  PROC DrawPart23()
    MoveL Offs(pOrigin,149.54,33.47,0.00),v40,z0,tPen\WObj:=wPaper;
    MoveL Offs(pOrigin,149.54,33.47,0.00),v40,z0,tPen\WObj:=wPaper;
    MoveL Offs(pOrigin,150.93,34.68,0.00),v40,z0,tPen\WObj:=wPaper;
    MoveL Offs(pOrigin,156.56,36.34,0.00),v40,fine,tPen\WObj:=wPaper;
    MoveL Offs(pOrigin,156.56,36.34,6.00),v60,z5,tPen\WObj:=wPaper;
    MoveL Offs(pOrigin,156.88,32.94,6.00),vTravel,z5,tPen\WObj:=wPaper;
    MoveL Offs(pOrigin,156.88,32.94,0.00),v60,z0,tPen\WObj:=wPaper;
    MoveL Offs(pOrigin,160.17,29.65,0.00),v40,z0,tPen\WObj:=wPaper;
    MoveL Offs(pOrigin,160.49,29.76,0.00),v40,z0,tPen\WObj:=wPaper;
    MoveL Offs(pOrigin,161.44,27.63,0.00),v40,z0,tPen\WObj:=wPaper;
    MoveL Offs(pOrigin,162.08,23.81,0.00),v40,z0,tPen\WObj:=wPaper;
    MoveL Offs(pOrigin,161.76,20.62,0.00),v40,z0,tPen\WObj:=wPaper;
    MoveL Offs(pOrigin,160.98,18.60,0.00),v40,z0,tPen\WObj:=wPaper;
    MoveL Offs(pOrigin,157.73,17.25,0.00),v40,z0,tPen\WObj:=wPaper;
    MoveL Offs(pOrigin,156.98,16.40,0.00),v40,z0,tPen\WObj:=wPaper;
    MoveL Offs(pOrigin,153.37,15.41,0.00),v40,z0,tPen\WObj:=wPaper;
    MoveL Offs(pOrigin,148.59,15.09,0.00),v40,z0,tPen\WObj:=wPaper;
    MoveL Offs(pOrigin,147.21,15.41,0.00),v40,fine,tPen\WObj:=wPaper;
    MoveL Offs(pOrigin,147.21,15.41,6.00),v60,z5,tPen\WObj:=wPaper;
    MoveL Offs(pOrigin,149.01,16.79,6.00),vTravel,z5,tPen\WObj:=wPaper;
    MoveL Offs(pOrigin,149.01,16.79,0.00),v60,z0,tPen\WObj:=wPaper;
    MoveL Offs(pOrigin,146.99,15.41,0.00),v40,z0,tPen\WObj:=wPaper;
    MoveL Offs(pOrigin,142.43,14.35,0.00),v40,z0,tPen\WObj:=wPaper;
    MoveL Offs(pOrigin,138.39,14.39,0.00),v40,z0,tPen\WObj:=wPaper;
    MoveL Offs(pOrigin,137.43,15.52,0.00),v40,z0,tPen\WObj:=wPaper;
    MoveL Offs(pOrigin,136.79,17.54,0.00),v40,z0,tPen\WObj:=wPaper;
    MoveL Offs(pOrigin,136.79,17.54,0.00),v40,z0,tPen\WObj:=wPaper;
    MoveL Offs(pOrigin,141.47,19.31,0.00),v40,z0,tPen\WObj:=wPaper;
    MoveL Offs(pOrigin,142.96,20.19,0.00),v40,z0,tPen\WObj:=wPaper;
    MoveL Offs(pOrigin,142.96,20.19,0.00),v40,z0,tPen\WObj:=wPaper;
    MoveL Offs(pOrigin,143.91,20.37,0.00),v40,z0,tPen\WObj:=wPaper;
    MoveL Offs(pOrigin,144.12,20.73,0.00),v40,z0,tPen\WObj:=wPaper;
    MoveL Offs(pOrigin,144.23,20.73,0.00),v40,z0,tPen\WObj:=wPaper;
    MoveL Offs(pOrigin,145.40,21.19,0.00),v40,z0,tPen\WObj:=wPaper;
    MoveL Offs(pOrigin,145.82,22.21,0.00),v40,z0,tPen\WObj:=wPaper;
    MoveL Offs(pOrigin,144.80,25.29,0.00),v40,z0,tPen\WObj:=wPaper;
    MoveL Offs(pOrigin,143.81,25.61,0.00),v40,z0,tPen\WObj:=wPaper;
    MoveL Offs(pOrigin,142.21,25.01,0.00),v40,z0,tPen\WObj:=wPaper;
    MoveL Offs(pOrigin,141.89,24.55,0.00),v40,z0,tPen\WObj:=wPaper;
    MoveL Offs(pOrigin,142.99,20.94,0.00),v40,z0,tPen\WObj:=wPaper;
    MoveL Offs(pOrigin,144.23,20.73,0.00),v40,z0,tPen\WObj:=wPaper;
    MoveL Offs(pOrigin,143.70,21.79,0.00),v40,z0,tPen\WObj:=wPaper;
    MoveL Offs(pOrigin,142.74,24.12,0.00),v40,z0,tPen\WObj:=wPaper;
    MoveL Offs(pOrigin,144.23,24.87,0.00),v40,fine,tPen\WObj:=wPaper;
    MoveL Offs(pOrigin,144.23,24.87,6.00),v60,z5,tPen\WObj:=wPaper;
    MoveL Offs(pOrigin,144.98,23.38,6.00),vTravel,z5,tPen\WObj:=wPaper;
    MoveL Offs(pOrigin,144.98,23.38,0.00),v60,z0,tPen\WObj:=wPaper;
    MoveL Offs(pOrigin,145.05,22.21,0.00),v40,z0,tPen\WObj:=wPaper;
    MoveL Offs(pOrigin,144.23,22.00,0.00),v40,fine,tPen\WObj:=wPaper;
    MoveL Offs(pOrigin,144.23,22.00,6.00),v60,z5,tPen\WObj:=wPaper;
    MoveL Offs(pOrigin,145.51,21.15,6.00),vTravel,z5,tPen\WObj:=wPaper;
    MoveL Offs(pOrigin,145.51,21.15,0.00),v60,z0,tPen\WObj:=wPaper;
    MoveL Offs(pOrigin,147.21,21.68,0.00),v40,fine,tPen\WObj:=wPaper;
    MoveL Offs(pOrigin,147.21,21.68,6.00),v60,z5,tPen\WObj:=wPaper;
    MoveL Offs(pOrigin,144.34,26.78,6.00),vTravel,z5,tPen\WObj:=wPaper;
    MoveL Offs(pOrigin,144.34,26.78,0.00),v60,z0,tPen\WObj:=wPaper;
    MoveL Offs(pOrigin,141.68,25.90,0.00),v40,z0,tPen\WObj:=wPaper;
    MoveL Offs(pOrigin,141.04,25.40,0.00),v40,z0,tPen\WObj:=wPaper;
    MoveL Offs(pOrigin,141.04,25.40,0.00),v40,z0,tPen\WObj:=wPaper;
    MoveL Offs(pOrigin,141.89,24.87,0.00),v40,z0,tPen\WObj:=wPaper;
    MoveL Offs(pOrigin,141.04,25.40,0.00),v40,z0,tPen\WObj:=wPaper;
    MoveL Offs(pOrigin,138.39,24.69,0.00),v40,z0,tPen\WObj:=wPaper;
    MoveL Offs(pOrigin,130.31,20.76,0.00),v40,z0,tPen\WObj:=wPaper;
    MoveL Offs(pOrigin,127.55,18.92,0.00),v40,z0,tPen\WObj:=wPaper;
    MoveL Offs(pOrigin,127.34,18.39,0.00),v40,z0,tPen\WObj:=wPaper;
    MoveL Offs(pOrigin,127.34,18.39,0.00),v40,z0,tPen\WObj:=wPaper;
    MoveL Offs(pOrigin,127.44,17.64,0.00),v40,z0,tPen\WObj:=wPaper;
    MoveL Offs(pOrigin,128.72,16.79,0.00),v40,z0,tPen\WObj:=wPaper;
    MoveL Offs(pOrigin,132.12,16.69,0.00),v40,z0,tPen\WObj:=wPaper;
    MoveL Offs(pOrigin,135.94,17.22,0.00),v40,z0,tPen\WObj:=wPaper;
    MoveL Offs(pOrigin,135.94,17.22,0.00),v40,z0,tPen\WObj:=wPaper;
    MoveL Offs(pOrigin,136.16,17.54,0.00),v40,z0,tPen\WObj:=wPaper;
    MoveL Offs(pOrigin,136.79,17.54,0.00),v40,z0,tPen\WObj:=wPaper;
    MoveL Offs(pOrigin,136.90,16.37,0.00),v40,z0,tPen\WObj:=wPaper;
    MoveL Offs(pOrigin,117.14,11.48,0.00),v40,z0,tPen\WObj:=wPaper;
    MoveL Offs(pOrigin,106.30,12.44,0.00),v40,z0,tPen\WObj:=wPaper;
    MoveL Offs(pOrigin,105.98,12.76,0.00),v40,z0,tPen\WObj:=wPaper;
    MoveL Offs(pOrigin,105.03,12.86,0.00),v40,z0,tPen\WObj:=wPaper;
    MoveL Offs(pOrigin,104.71,13.18,0.00),v40,z0,tPen\WObj:=wPaper;
    MoveL Offs(pOrigin,104.28,12.97,0.00),v40,z0,tPen\WObj:=wPaper;
    MoveL Offs(pOrigin,105.03,12.86,0.00),v40,z0,tPen\WObj:=wPaper;
    MoveL Offs(pOrigin,105.77,12.76,0.00),v40,z0,tPen\WObj:=wPaper;
    MoveL Offs(pOrigin,107.57,13.39,0.00),v40,z0,tPen\WObj:=wPaper;
    MoveL Offs(pOrigin,124.15,16.90,0.00),v40,z0,tPen\WObj:=wPaper;
    MoveL Offs(pOrigin,125.21,17.54,0.00),v40,z0,tPen\WObj:=wPaper;
    MoveL Offs(pOrigin,125.21,17.54,0.00),v40,z0,tPen\WObj:=wPaper;
    MoveL Offs(pOrigin,122.88,18.21,0.00),v40,z0,tPen\WObj:=wPaper;
    MoveL Offs(pOrigin,122.34,19.88,0.00),v40,fine,tPen\WObj:=wPaper;
    MoveL Offs(pOrigin,122.34,19.88,6.00),v60,z5,tPen\WObj:=wPaper;
    MoveL Offs(pOrigin,123.09,21.15,6.00),vTravel,z5,tPen\WObj:=wPaper;
    MoveL Offs(pOrigin,123.09,21.15,0.00),v60,z0,tPen\WObj:=wPaper;
    MoveL Offs(pOrigin,123.51,21.58,0.00),v40,z0,tPen\WObj:=wPaper;
    MoveL Offs(pOrigin,123.09,21.15,0.00),v40,fine,tPen\WObj:=wPaper;
    MoveL Offs(pOrigin,123.09,21.15,6.00),v60,z5,tPen\WObj:=wPaper;
    MoveL Offs(pOrigin,124.57,22.42,6.00),vTravel,z5,tPen\WObj:=wPaper;
    MoveL Offs(pOrigin,124.57,22.42,0.00),v60,z0,tPen\WObj:=wPaper;
    MoveL Offs(pOrigin,125.00,22.85,0.00),v40,z0,tPen\WObj:=wPaper;
    MoveL Offs(pOrigin,124.57,22.42,0.00),v40,fine,tPen\WObj:=wPaper;
    MoveL Offs(pOrigin,124.57,22.42,6.00),v60,z5,tPen\WObj:=wPaper;
    MoveL Offs(pOrigin,121.07,22.32,6.00),vTravel,z5,tPen\WObj:=wPaper;
    MoveL Offs(pOrigin,121.07,22.32,0.00),v60,z0,tPen\WObj:=wPaper;
    MoveL Offs(pOrigin,119.37,22.42,0.00),v40,fine,tPen\WObj:=wPaper;
    MoveL Offs(pOrigin,119.37,22.42,6.00),v60,z5,tPen\WObj:=wPaper;
    MoveL Offs(pOrigin,112.99,23.70,6.00),vTravel,z5,tPen\WObj:=wPaper;
    MoveL Offs(pOrigin,112.99,23.70,0.00),v60,z0,tPen\WObj:=wPaper;
    MoveL Offs(pOrigin,111.82,24.23,0.00),v40,z0,tPen\WObj:=wPaper;
    MoveL Offs(pOrigin,112.36,24.76,0.00),v40,z0,tPen\WObj:=wPaper;
    MoveL Offs(pOrigin,111.61,24.27,0.00),v40,z0,tPen\WObj:=wPaper;
    MoveL Offs(pOrigin,109.70,25.01,0.00),v40,z0,tPen\WObj:=wPaper;
    MoveL Offs(pOrigin,107.93,26.36,0.00),v40,z0,tPen\WObj:=wPaper;
    MoveL Offs(pOrigin,106.72,28.48,0.00),v40,z0,tPen\WObj:=wPaper;
    MoveL Offs(pOrigin,106.72,28.48,0.00),v40,z0,tPen\WObj:=wPaper;
    MoveL Offs(pOrigin,100.88,31.49,0.00),v40,z0,tPen\WObj:=wPaper;
    MoveL Offs(pOrigin,93.44,33.86,0.00),v40,z0,tPen\WObj:=wPaper;
    MoveL Offs(pOrigin,91.85,34.75,0.00),v40,fine,tPen\WObj:=wPaper;
    MoveL Offs(pOrigin,91.85,34.75,6.00),v60,z5,tPen\WObj:=wPaper;
    MoveL Offs(pOrigin,90.79,28.59,6.00),vTravel,z5,tPen\WObj:=wPaper;
    MoveL Offs(pOrigin,90.79,28.59,0.00),v60,z0,tPen\WObj:=wPaper;
    MoveL Offs(pOrigin,94.61,26.67,0.00),v40,z0,tPen\WObj:=wPaper;
    MoveL Offs(pOrigin,94.61,26.67,0.00),v40,z0,tPen\WObj:=wPaper;
  ENDPROC

  PROC DrawPart24()
    MoveL Offs(pOrigin,94.08,25.19,0.00),v40,z0,tPen\WObj:=wPaper;
    MoveL Offs(pOrigin,94.08,25.19,0.00),v40,z0,tPen\WObj:=wPaper;
    MoveL Offs(pOrigin,95.04,24.87,0.00),v40,z0,tPen\WObj:=wPaper;
    MoveL Offs(pOrigin,95.04,24.87,0.00),v40,z0,tPen\WObj:=wPaper;
    MoveL Offs(pOrigin,95.57,26.36,0.00),v40,z0,tPen\WObj:=wPaper;
    MoveL Offs(pOrigin,95.57,26.36,0.00),v40,z0,tPen\WObj:=wPaper;
    MoveL Offs(pOrigin,104.49,23.91,0.00),v40,z0,tPen\WObj:=wPaper;
    MoveL Offs(pOrigin,104.81,23.59,0.00),v40,fine,tPen\WObj:=wPaper;
    MoveL Offs(pOrigin,104.81,23.59,6.00),v60,z5,tPen\WObj:=wPaper;
    MoveL Offs(pOrigin,109.06,23.27,6.00),vTravel,z5,tPen\WObj:=wPaper;
    MoveL Offs(pOrigin,109.06,23.27,0.00),v60,z0,tPen\WObj:=wPaper;
    MoveL Offs(pOrigin,109.59,24.98,0.00),v40,fine,tPen\WObj:=wPaper;
    MoveL Offs(pOrigin,109.59,24.98,6.00),v60,z5,tPen\WObj:=wPaper;
    MoveL Offs(pOrigin,117.56,29.54,6.00),vTravel,z5,tPen\WObj:=wPaper;
    MoveL Offs(pOrigin,117.56,29.54,0.00),v60,z0,tPen\WObj:=wPaper;
    MoveL Offs(pOrigin,113.31,35.49,0.00),v40,z0,tPen\WObj:=wPaper;
    MoveL Offs(pOrigin,113.42,36.13,0.00),v40,z0,tPen\WObj:=wPaper;
    MoveL Offs(pOrigin,115.44,35.53,0.00),v40,z0,tPen\WObj:=wPaper;
    MoveL Offs(pOrigin,117.67,34.11,0.00),v40,fine,tPen\WObj:=wPaper;
    MoveL Offs(pOrigin,117.67,34.11,6.00),v60,z5,tPen\WObj:=wPaper;
    MoveL Offs(pOrigin,118.41,39.00,6.00),vTravel,z5,tPen\WObj:=wPaper;
    MoveL Offs(pOrigin,118.41,39.00,0.00),v60,z0,tPen\WObj:=wPaper;
    MoveL Offs(pOrigin,115.01,44.10,0.00),v40,fine,tPen\WObj:=wPaper;
    MoveL Offs(pOrigin,115.01,44.10,6.00),v60,z5,tPen\WObj:=wPaper;
    MoveL Offs(pOrigin,123.09,37.51,6.00),vTravel,z5,tPen\WObj:=wPaper;
    MoveL Offs(pOrigin,123.09,37.51,0.00),v60,z0,tPen\WObj:=wPaper;
    MoveL Offs(pOrigin,122.77,36.56,0.00),v40,z0,tPen\WObj:=wPaper;
    MoveL Offs(pOrigin,123.19,35.74,0.00),v40,z0,tPen\WObj:=wPaper;
    MoveL Offs(pOrigin,124.26,35.28,0.00),v40,z0,tPen\WObj:=wPaper;
    MoveL Offs(pOrigin,125.32,35.81,0.00),v40,z0,tPen\WObj:=wPaper;
    MoveL Offs(pOrigin,125.64,36.88,0.00),v40,z0,tPen\WObj:=wPaper;
    MoveL Offs(pOrigin,125.11,37.83,0.00),v40,z0,tPen\WObj:=wPaper;
    MoveL Offs(pOrigin,124.04,38.15,0.00),v40,z0,tPen\WObj:=wPaper;
    MoveL Offs(pOrigin,123.09,37.51,0.00),v40,fine,tPen\WObj:=wPaper;
    MoveL Offs(pOrigin,123.09,37.51,6.00),v60,z5,tPen\WObj:=wPaper;
    MoveL Offs(pOrigin,126.59,28.48,6.00),vTravel,z5,tPen\WObj:=wPaper;
    MoveL Offs(pOrigin,126.59,28.48,0.00),v60,z0,tPen\WObj:=wPaper;
    MoveL Offs(pOrigin,126.91,28.80,0.00),v40,z0,tPen\WObj:=wPaper;
    MoveL Offs(pOrigin,126.59,28.48,0.00),v40,fine,tPen\WObj:=wPaper;
    MoveL Offs(pOrigin,126.59,28.48,6.00),v60,z5,tPen\WObj:=wPaper;
    MoveL Offs(pOrigin,124.68,26.57,6.00),vTravel,z5,tPen\WObj:=wPaper;
    MoveL Offs(pOrigin,124.68,26.57,0.00),v60,z0,tPen\WObj:=wPaper;
    MoveL Offs(pOrigin,125.11,26.99,0.00),v40,z0,tPen\WObj:=wPaper;
    MoveL Offs(pOrigin,124.68,26.57,0.00),v40,fine,tPen\WObj:=wPaper;
    MoveL Offs(pOrigin,124.68,26.57,6.00),v60,z5,tPen\WObj:=wPaper;
    MoveL Offs(pOrigin,127.34,18.39,6.00),vTravel,z5,tPen\WObj:=wPaper;
    MoveL Offs(pOrigin,127.34,18.39,0.00),v60,z0,tPen\WObj:=wPaper;
    MoveL Offs(pOrigin,126.38,18.21,0.00),v40,z0,tPen\WObj:=wPaper;
    MoveL Offs(pOrigin,125.64,17.54,0.00),v40,z0,tPen\WObj:=wPaper;
    MoveL Offs(pOrigin,125.64,17.54,0.00),v40,z0,tPen\WObj:=wPaper;
    MoveL Offs(pOrigin,127.34,17.64,0.00),v40,z0,tPen\WObj:=wPaper;
    MoveL Offs(pOrigin,127.87,17.11,0.00),v40,z0,tPen\WObj:=wPaper;
    MoveL Offs(pOrigin,127.55,17.43,0.00),v40,z0,tPen\WObj:=wPaper;
    MoveL Offs(pOrigin,127.87,17.11,0.00),v40,fine,tPen\WObj:=wPaper;
    MoveL Offs(pOrigin,127.87,17.11,6.00),v60,z5,tPen\WObj:=wPaper;
    MoveL Offs(pOrigin,137.43,15.41,6.00),vTravel,z5,tPen\WObj:=wPaper;
    MoveL Offs(pOrigin,137.43,15.41,0.00),v60,z0,tPen\WObj:=wPaper;
    MoveL Offs(pOrigin,116.71,9.99,0.00),v40,z0,tPen\WObj:=wPaper;
    MoveL Offs(pOrigin,104.71,11.06,0.00),v40,z0,tPen\WObj:=wPaper;
    MoveL Offs(pOrigin,104.49,11.69,0.00),v40,z0,tPen\WObj:=wPaper;
    MoveL Offs(pOrigin,105.03,12.86,0.00),v40,fine,tPen\WObj:=wPaper;
    MoveL Offs(pOrigin,105.03,12.86,6.00),v60,z5,tPen\WObj:=wPaper;
    MoveL Offs(pOrigin,104.49,11.06,6.00),vTravel,z5,tPen\WObj:=wPaper;
    MoveL Offs(pOrigin,104.49,11.06,0.00),v60,z0,tPen\WObj:=wPaper;
    MoveL Offs(pOrigin,104.71,9.68,0.00),v40,z0,tPen\WObj:=wPaper;
    MoveL Offs(pOrigin,103.54,9.46,0.00),v40,z0,tPen\WObj:=wPaper;
    MoveL Offs(pOrigin,106.41,9.68,0.00),v40,z0,tPen\WObj:=wPaper;
    MoveL Offs(pOrigin,116.07,8.61,0.00),v40,z0,tPen\WObj:=wPaper;
    MoveL Offs(pOrigin,117.56,8.72,0.00),v40,z0,tPen\WObj:=wPaper;
    MoveL Offs(pOrigin,138.28,14.35,0.00),v40,fine,tPen\WObj:=wPaper;
    MoveL Offs(pOrigin,138.28,14.35,6.00),v60,z5,tPen\WObj:=wPaper;
    MoveL Offs(pOrigin,157.09,16.37,6.00),vTravel,z5,tPen\WObj:=wPaper;
    MoveL Offs(pOrigin,157.09,16.37,0.00),v60,z0,tPen\WObj:=wPaper;
    MoveL Offs(pOrigin,158.36,15.94,0.00),v40,z0,tPen\WObj:=wPaper;
    MoveL Offs(pOrigin,158.36,15.94,0.00),v40,z0,tPen\WObj:=wPaper;
    MoveL Offs(pOrigin,158.79,15.41,0.00),v40,z0,tPen\WObj:=wPaper;
    MoveL Offs(pOrigin,160.49,15.31,0.00),v40,z0,tPen\WObj:=wPaper;
    MoveL Offs(pOrigin,167.50,16.26,0.00),v40,fine,tPen\WObj:=wPaper;
    MoveL Offs(pOrigin,167.50,16.26,6.00),v60,z5,tPen\WObj:=wPaper;
    MoveL Offs(pOrigin,161.02,18.49,6.00),vTravel,z5,tPen\WObj:=wPaper;
    MoveL Offs(pOrigin,161.02,18.49,0.00),v60,z0,tPen\WObj:=wPaper;
    MoveL Offs(pOrigin,160.84,17.54,0.00),v40,z0,tPen\WObj:=wPaper;
    MoveL Offs(pOrigin,160.06,16.58,0.00),v40,z0,tPen\WObj:=wPaper;
    MoveL Offs(pOrigin,158.36,15.94,0.00),v40,fine,tPen\WObj:=wPaper;
    MoveL Offs(pOrigin,158.36,15.94,6.00),v60,z5,tPen\WObj:=wPaper;
    MoveL Offs(pOrigin,161.34,22.74,6.00),vTravel,z5,tPen\WObj:=wPaper;
    MoveL Offs(pOrigin,161.34,22.74,0.00),v60,z0,tPen\WObj:=wPaper;
    MoveL Offs(pOrigin,161.34,24.55,0.00),v40,z0,tPen\WObj:=wPaper;
    MoveL Offs(pOrigin,160.63,27.31,0.00),v40,z0,tPen\WObj:=wPaper;
    MoveL Offs(pOrigin,158.68,30.71,0.00),v40,fine,tPen\WObj:=wPaper;
    MoveL Offs(pOrigin,158.68,30.71,6.00),v60,z5,tPen\WObj:=wPaper;
    MoveL Offs(pOrigin,160.49,29.76,6.00),vTravel,z5,tPen\WObj:=wPaper;
    MoveL Offs(pOrigin,160.49,29.76,0.00),v60,z0,tPen\WObj:=wPaper;
    MoveL Offs(pOrigin,160.45,30.29,0.00),v40,z0,tPen\WObj:=wPaper;
    MoveL Offs(pOrigin,159.32,31.99,0.00),v40,z0,tPen\WObj:=wPaper;
    MoveL Offs(pOrigin,156.98,33.65,0.00),v40,z0,tPen\WObj:=wPaper;
    MoveL Offs(pOrigin,155.07,34.22,0.00),v40,z0,tPen\WObj:=wPaper;
    MoveL Offs(pOrigin,153.26,34.22,0.00),v40,z0,tPen\WObj:=wPaper;
    MoveL Offs(pOrigin,151.24,33.65,0.00),v40,z0,tPen\WObj:=wPaper;
    MoveL Offs(pOrigin,150.93,33.16,0.00),v40,z0,tPen\WObj:=wPaper;
    MoveL Offs(pOrigin,150.93,33.16,0.00),v40,z0,tPen\WObj:=wPaper;
    MoveL Offs(pOrigin,151.24,32.84,0.00),v40,z0,tPen\WObj:=wPaper;
    MoveL Offs(pOrigin,152.84,32.66,0.00),v40,z0,tPen\WObj:=wPaper;
    MoveL Offs(pOrigin,155.28,33.05,0.00),v40,z0,tPen\WObj:=wPaper;
    MoveL Offs(pOrigin,155.28,33.05,0.00),v40,z0,tPen\WObj:=wPaper;
    MoveL Offs(pOrigin,156.88,32.94,0.00),v40,fine,tPen\WObj:=wPaper;
    MoveL Offs(pOrigin,156.88,32.94,6.00),v60,z5,tPen\WObj:=wPaper;
    MoveL Offs(pOrigin,150.93,33.16,6.00),vTravel,z5,tPen\WObj:=wPaper;
    MoveL Offs(pOrigin,150.93,33.16,0.00),v60,z0,tPen\WObj:=wPaper;
    MoveL Offs(pOrigin,149.54,33.47,0.00),v40,fine,tPen\WObj:=wPaper;
    MoveL Offs(pOrigin,149.54,33.47,6.00),v60,z5,tPen\WObj:=wPaper;
    MoveL Offs(pOrigin,147.21,35.28,6.00),vTravel,z5,tPen\WObj:=wPaper;
    MoveL Offs(pOrigin,147.21,35.28,0.00),v60,z0,tPen\WObj:=wPaper;
    MoveL Offs(pOrigin,146.14,41.23,0.00),v40,z0,tPen\WObj:=wPaper;
    MoveL Offs(pOrigin,146.25,51.11,0.00),v40,z0,tPen\WObj:=wPaper;
    MoveL Offs(pOrigin,145.93,51.54,0.00),v40,fine,tPen\WObj:=wPaper;
    MoveL Offs(pOrigin,145.93,51.54,6.00),v60,z5,tPen\WObj:=wPaper;
    MoveL Offs(pOrigin,174.94,48.67,6.00),vTravel,z5,tPen\WObj:=wPaper;
    MoveL Offs(pOrigin,174.94,48.67,0.00),v60,z0,tPen\WObj:=wPaper;
    MoveL Offs(pOrigin,176.11,47.71,0.00),v40,fine,tPen\WObj:=wPaper;
  ENDPROC

  PROC DrawPart25()
    MoveL Offs(pOrigin,176.11,47.71,6.00),v60,z5,tPen\WObj:=wPaper;
    MoveL Offs(pOrigin,180.89,52.60,6.00),vTravel,z5,tPen\WObj:=wPaper;
    MoveL Offs(pOrigin,180.89,52.60,0.00),v60,z0,tPen\WObj:=wPaper;
    MoveL Offs(pOrigin,181.21,52.92,0.00),v40,z0,tPen\WObj:=wPaper;
    MoveL Offs(pOrigin,180.89,52.60,0.00),v40,fine,tPen\WObj:=wPaper;
    MoveL Offs(pOrigin,180.89,52.60,6.00),v60,z5,tPen\WObj:=wPaper;
    MoveL Offs(pOrigin,198.63,56.64,6.00),vTravel,z5,tPen\WObj:=wPaper;
    MoveL Offs(pOrigin,198.63,56.64,0.00),v60,z0,tPen\WObj:=wPaper;
    MoveL Offs(pOrigin,200.44,55.58,0.00),v40,fine,tPen\WObj:=wPaper;
    MoveL Offs(pOrigin,200.44,55.58,6.00),v60,z5,tPen\WObj:=wPaper;
    MoveL Offs(pOrigin,169.73,31.03,6.00),vTravel,z5,tPen\WObj:=wPaper;
    MoveL Offs(pOrigin,169.73,31.03,0.00),v60,z0,tPen\WObj:=wPaper;
    MoveL Offs(pOrigin,168.88,31.88,0.00),v40,z0,tPen\WObj:=wPaper;
    MoveL Offs(pOrigin,169.73,31.03,0.00),v40,fine,tPen\WObj:=wPaper;
    MoveL Offs(pOrigin,169.73,31.03,6.00),v60,z5,tPen\WObj:=wPaper;
    MoveL Offs(pOrigin,168.77,31.99,6.00),vTravel,z5,tPen\WObj:=wPaper;
    MoveL Offs(pOrigin,168.77,31.99,0.00),v60,z0,tPen\WObj:=wPaper;
    MoveL Offs(pOrigin,168.46,32.31,0.00),v40,z0,tPen\WObj:=wPaper;
    MoveL Offs(pOrigin,168.77,31.99,0.00),v40,fine,tPen\WObj:=wPaper;
    MoveL Offs(pOrigin,168.77,31.99,6.00),v60,z5,tPen\WObj:=wPaper;
    MoveL Offs(pOrigin,167.39,31.14,6.00),vTravel,z5,tPen\WObj:=wPaper;
    MoveL Offs(pOrigin,167.39,31.14,0.00),v60,z0,tPen\WObj:=wPaper;
    MoveL Offs(pOrigin,168.99,28.48,0.00),v40,fine,tPen\WObj:=wPaper;
    MoveL Offs(pOrigin,168.99,28.48,6.00),v60,z5,tPen\WObj:=wPaper;
    MoveL Offs(pOrigin,100.35,20.51,6.00),vTravel,z5,tPen\WObj:=wPaper;
    MoveL Offs(pOrigin,100.35,20.51,0.00),v60,z0,tPen\WObj:=wPaper;
    MoveL Offs(pOrigin,99.71,19.34,0.00),v40,fine,tPen\WObj:=wPaper;
    MoveL Offs(pOrigin,99.71,19.34,6.00),v60,z5,tPen\WObj:=wPaper;
    MoveL Offs(pOrigin,100.35,20.51,6.00),vTravel,z5,tPen\WObj:=wPaper;
    MoveL Offs(pOrigin,100.35,20.51,0.00),v60,z0,tPen\WObj:=wPaper;
    MoveL Offs(pOrigin,97.06,20.73,0.00),v40,z0,tPen\WObj:=wPaper;
    MoveL Offs(pOrigin,94.61,21.47,0.00),v40,z0,tPen\WObj:=wPaper;
    MoveL Offs(pOrigin,94.61,21.47,0.00),v40,z0,tPen\WObj:=wPaper;
    MoveL Offs(pOrigin,95.78,23.17,0.00),v40,z0,tPen\WObj:=wPaper;
    MoveL Offs(pOrigin,95.60,24.12,0.00),v40,z0,tPen\WObj:=wPaper;
    MoveL Offs(pOrigin,95.04,24.87,0.00),v40,z0,tPen\WObj:=wPaper;
    MoveL Offs(pOrigin,95.04,24.12,0.00),v40,z0,tPen\WObj:=wPaper;
    MoveL Offs(pOrigin,93.76,24.55,0.00),v40,z0,tPen\WObj:=wPaper;
    MoveL Offs(pOrigin,93.12,24.12,0.00),v40,fine,tPen\WObj:=wPaper;
    MoveL Offs(pOrigin,93.12,24.12,6.00),v60,z5,tPen\WObj:=wPaper;
    MoveL Offs(pOrigin,94.08,25.19,6.00),vTravel,z5,tPen\WObj:=wPaper;
    MoveL Offs(pOrigin,94.08,25.19,0.00),v60,z0,tPen\WObj:=wPaper;
    MoveL Offs(pOrigin,93.12,24.76,0.00),v40,z0,tPen\WObj:=wPaper;
    MoveL Offs(pOrigin,92.56,24.02,0.00),v40,z0,tPen\WObj:=wPaper;
    MoveL Offs(pOrigin,92.59,22.11,0.00),v40,z0,tPen\WObj:=wPaper;
    MoveL Offs(pOrigin,92.59,22.11,0.00),v40,z0,tPen\WObj:=wPaper;
    MoveL Offs(pOrigin,93.55,21.58,0.00),v40,z0,tPen\WObj:=wPaper;
    MoveL Offs(pOrigin,94.61,21.47,0.00),v40,fine,tPen\WObj:=wPaper;
    MoveL Offs(pOrigin,94.61,21.47,6.00),v60,z5,tPen\WObj:=wPaper;
    MoveL Offs(pOrigin,92.59,22.11,6.00),vTravel,z5,tPen\WObj:=wPaper;
    MoveL Offs(pOrigin,92.59,22.11,0.00),v60,z0,tPen\WObj:=wPaper;
    MoveL Offs(pOrigin,89.62,23.17,0.00),v40,fine,tPen\WObj:=wPaper;
    MoveL Offs(pOrigin,89.62,23.17,6.00),v60,z5,tPen\WObj:=wPaper;
    MoveL Offs(pOrigin,94.61,26.67,6.00),vTravel,z5,tPen\WObj:=wPaper;
    MoveL Offs(pOrigin,94.61,26.67,0.00),v60,z0,tPen\WObj:=wPaper;
    MoveL Offs(pOrigin,95.57,26.36,0.00),v40,fine,tPen\WObj:=wPaper;
    MoveL Offs(pOrigin,95.57,26.36,6.00),v60,z5,tPen\WObj:=wPaper;
    MoveL Offs(pOrigin,97.27,13.29,6.00),vTravel,z5,tPen\WObj:=wPaper;
    MoveL Offs(pOrigin,97.27,13.29,0.00),v60,z0,tPen\WObj:=wPaper;
    MoveL Offs(pOrigin,93.34,13.93,0.00),v40,z0,tPen\WObj:=wPaper;
    MoveL Offs(pOrigin,44.04,18.71,0.00),v40,fine,tPen\WObj:=wPaper;
    MoveL Offs(pOrigin,44.04,18.71,6.00),v60,z5,tPen\WObj:=wPaper;
    MoveL Offs(pOrigin,49.46,19.45,6.00),vTravel,z5,tPen\WObj:=wPaper;
    MoveL Offs(pOrigin,49.46,19.45,0.00),v60,z0,tPen\WObj:=wPaper;
    MoveL Offs(pOrigin,64.54,21.26,0.00),v40,z0,tPen\WObj:=wPaper;
    MoveL Offs(pOrigin,65.71,21.79,0.00),v40,fine,tPen\WObj:=wPaper;
    MoveL Offs(pOrigin,65.71,21.79,6.00),v60,z5,tPen\WObj:=wPaper;
    MoveL Offs(pOrigin,69.86,25.40,6.00),vTravel,z5,tPen\WObj:=wPaper;
    MoveL Offs(pOrigin,69.86,25.40,0.00),v60,z0,tPen\WObj:=wPaper;
    MoveL Offs(pOrigin,70.39,24.23,0.00),v40,z0,tPen\WObj:=wPaper;
    MoveL Offs(pOrigin,71.45,23.06,0.00),v40,z0,tPen\WObj:=wPaper;
    MoveL Offs(pOrigin,71.66,22.96,0.00),v40,z0,tPen\WObj:=wPaper;
    MoveL Offs(pOrigin,73.36,22.11,0.00),v40,z0,tPen\WObj:=wPaper;
    MoveL Offs(pOrigin,74.85,22.00,0.00),v40,z0,tPen\WObj:=wPaper;
    MoveL Offs(pOrigin,75.17,22.32,0.00),v40,fine,tPen\WObj:=wPaper;
    MoveL Offs(pOrigin,75.17,22.32,6.00),v60,z5,tPen\WObj:=wPaper;
    MoveL Offs(pOrigin,77.19,21.26,6.00),vTravel,z5,tPen\WObj:=wPaper;
    MoveL Offs(pOrigin,77.19,21.26,0.00),v60,z0,tPen\WObj:=wPaper;
    MoveL Offs(pOrigin,74.74,20.73,0.00),v40,z0,tPen\WObj:=wPaper;
    MoveL Offs(pOrigin,71.45,20.94,0.00),v40,fine,tPen\WObj:=wPaper;
    MoveL Offs(pOrigin,71.45,20.94,6.00),v60,z5,tPen\WObj:=wPaper;
    MoveL Offs(pOrigin,71.45,25.29,6.00),vTravel,z5,tPen\WObj:=wPaper;
    MoveL Offs(pOrigin,71.45,25.29,0.00),v60,z0,tPen\WObj:=wPaper;
    MoveL Offs(pOrigin,71.24,27.74,0.00),v40,z0,tPen\WObj:=wPaper;
    MoveL Offs(pOrigin,73.01,31.99,0.00),v40,z0,tPen\WObj:=wPaper;
    MoveL Offs(pOrigin,75.49,34.96,0.00),v40,z0,tPen\WObj:=wPaper;
    MoveL Offs(pOrigin,78.89,36.98,0.00),v40,z0,tPen\WObj:=wPaper;
    MoveL Offs(pOrigin,78.89,36.98,0.00),v40,z0,tPen\WObj:=wPaper;
    MoveL Offs(pOrigin,81.54,37.09,0.00),v40,z0,tPen\WObj:=wPaper;
    MoveL Offs(pOrigin,81.54,37.09,0.00),v40,z0,tPen\WObj:=wPaper;
    MoveL Offs(pOrigin,81.30,37.69,0.00),v40,z0,tPen\WObj:=wPaper;
    MoveL Offs(pOrigin,79.84,38.15,0.00),v40,z0,tPen\WObj:=wPaper;
    MoveL Offs(pOrigin,77.72,38.04,0.00),v40,z0,tPen\WObj:=wPaper;
    MoveL Offs(pOrigin,76.55,37.51,0.00),v40,z0,tPen\WObj:=wPaper;
    MoveL Offs(pOrigin,76.55,37.51,0.00),v40,z0,tPen\WObj:=wPaper;
    MoveL Offs(pOrigin,75.17,37.02,0.00),v40,z0,tPen\WObj:=wPaper;
    MoveL Offs(pOrigin,71.45,34.61,0.00),v40,z0,tPen\WObj:=wPaper;
    MoveL Offs(pOrigin,69.96,33.16,0.00),v40,z0,tPen\WObj:=wPaper;
    MoveL Offs(pOrigin,68.97,31.77,0.00),v40,z0,tPen\WObj:=wPaper;
    MoveL Offs(pOrigin,68.26,29.86,0.00),v40,z0,tPen\WObj:=wPaper;
    MoveL Offs(pOrigin,68.26,28.16,0.00),v40,z0,tPen\WObj:=wPaper;
    MoveL Offs(pOrigin,68.58,27.63,0.00),v40,z0,tPen\WObj:=wPaper;
    MoveL Offs(pOrigin,68.58,27.63,0.00),v40,z0,tPen\WObj:=wPaper;
    MoveL Offs(pOrigin,69.18,25.72,0.00),v40,z0,tPen\WObj:=wPaper;
    MoveL Offs(pOrigin,69.86,25.40,0.00),v40,fine,tPen\WObj:=wPaper;
    MoveL Offs(pOrigin,69.86,25.40,6.00),v60,z5,tPen\WObj:=wPaper;
    MoveL Offs(pOrigin,68.58,27.63,6.00),vTravel,z5,tPen\WObj:=wPaper;
    MoveL Offs(pOrigin,68.58,27.63,0.00),v60,z0,tPen\WObj:=wPaper;
    MoveL Offs(pOrigin,69.32,28.27,0.00),v40,z0,tPen\WObj:=wPaper;
    MoveL Offs(pOrigin,69.32,28.27,0.00),v40,z0,tPen\WObj:=wPaper;
    MoveL Offs(pOrigin,70.07,28.91,0.00),v40,z0,tPen\WObj:=wPaper;
    MoveL Offs(pOrigin,70.07,29.12,0.00),v40,z0,tPen\WObj:=wPaper;
    MoveL Offs(pOrigin,70.78,29.01,0.00),v40,z0,tPen\WObj:=wPaper;
    MoveL Offs(pOrigin,72.26,32.41,0.00),v40,z0,tPen\WObj:=wPaper;
    MoveL Offs(pOrigin,74.11,34.64,0.00),v40,z0,tPen\WObj:=wPaper;
    MoveL Offs(pOrigin,74.32,34.96,0.00),v40,z0,tPen\WObj:=wPaper;
    MoveL Offs(pOrigin,75.06,35.39,0.00),v40,z0,tPen\WObj:=wPaper;
    MoveL Offs(pOrigin,74.96,35.71,0.00),v40,fine,tPen\WObj:=wPaper;
    MoveL Offs(pOrigin,74.96,35.71,6.00),v60,z5,tPen\WObj:=wPaper;
    MoveL Offs(pOrigin,76.76,36.98,6.00),vTravel,z5,tPen\WObj:=wPaper;
  ENDPROC

  PROC DrawPart26()
    MoveL Offs(pOrigin,76.76,36.98,0.00),v60,z0,tPen\WObj:=wPaper;
    MoveL Offs(pOrigin,73.89,35.07,0.00),v40,z0,tPen\WObj:=wPaper;
    MoveL Offs(pOrigin,72.30,33.58,0.00),v40,z0,tPen\WObj:=wPaper;
    MoveL Offs(pOrigin,71.98,33.47,0.00),v40,z0,tPen\WObj:=wPaper;
    MoveL Offs(pOrigin,72.30,34.86,0.00),v40,z0,tPen\WObj:=wPaper;
    MoveL Offs(pOrigin,73.04,34.22,0.00),v40,z0,tPen\WObj:=wPaper;
    MoveL Offs(pOrigin,73.47,34.64,0.00),v40,z0,tPen\WObj:=wPaper;
    MoveL Offs(pOrigin,73.04,34.22,0.00),v40,z0,tPen\WObj:=wPaper;
    MoveL Offs(pOrigin,73.26,33.69,0.00),v40,z0,tPen\WObj:=wPaper;
    MoveL Offs(pOrigin,73.57,34.01,0.00),v40,z0,tPen\WObj:=wPaper;
    MoveL Offs(pOrigin,73.26,33.69,0.00),v40,fine,tPen\WObj:=wPaper;
    MoveL Offs(pOrigin,73.26,33.69,6.00),v60,z5,tPen\WObj:=wPaper;
    MoveL Offs(pOrigin,71.56,32.62,6.00),vTravel,z5,tPen\WObj:=wPaper;
    MoveL Offs(pOrigin,71.56,32.62,0.00),v60,z0,tPen\WObj:=wPaper;
    MoveL Offs(pOrigin,71.03,31.67,0.00),v40,z0,tPen\WObj:=wPaper;
    MoveL Offs(pOrigin,71.03,31.67,0.00),v40,z0,tPen\WObj:=wPaper;
    MoveL Offs(pOrigin,70.49,30.71,0.00),v40,z0,tPen\WObj:=wPaper;
    MoveL Offs(pOrigin,70.28,31.03,0.00),v40,z0,tPen\WObj:=wPaper;
    MoveL Offs(pOrigin,70.39,31.67,0.00),v40,z0,tPen\WObj:=wPaper;
    MoveL Offs(pOrigin,70.81,31.88,0.00),v40,fine,tPen\WObj:=wPaper;
    MoveL Offs(pOrigin,70.81,31.88,6.00),v60,z5,tPen\WObj:=wPaper;
    MoveL Offs(pOrigin,70.71,33.79,6.00),vTravel,z5,tPen\WObj:=wPaper;
    MoveL Offs(pOrigin,70.71,33.79,0.00),v60,z0,tPen\WObj:=wPaper;
    MoveL Offs(pOrigin,71.13,34.22,0.00),v40,z0,tPen\WObj:=wPaper;
    MoveL Offs(pOrigin,70.71,33.79,0.00),v40,fine,tPen\WObj:=wPaper;
    MoveL Offs(pOrigin,70.71,33.79,6.00),v60,z5,tPen\WObj:=wPaper;
    MoveL Offs(pOrigin,70.28,29.86,6.00),vTravel,z5,tPen\WObj:=wPaper;
    MoveL Offs(pOrigin,70.28,29.86,0.00),v60,z0,tPen\WObj:=wPaper;
    MoveL Offs(pOrigin,69.64,29.76,0.00),v40,z0,tPen\WObj:=wPaper;
    MoveL Offs(pOrigin,70.18,29.54,0.00),v40,z0,tPen\WObj:=wPaper;
    MoveL Offs(pOrigin,69.54,29.23,0.00),v40,z0,tPen\WObj:=wPaper;
    MoveL Offs(pOrigin,69.22,28.91,0.00),v40,z0,tPen\WObj:=wPaper;
    MoveL Offs(pOrigin,69.32,28.27,0.00),v40,fine,tPen\WObj:=wPaper;
    MoveL Offs(pOrigin,69.32,28.27,6.00),v60,z5,tPen\WObj:=wPaper;
    MoveL Offs(pOrigin,71.24,27.95,6.00),vTravel,z5,tPen\WObj:=wPaper;
    MoveL Offs(pOrigin,71.24,27.95,0.00),v60,z0,tPen\WObj:=wPaper;
    MoveL Offs(pOrigin,70.64,28.06,0.00),v40,z0,tPen\WObj:=wPaper;
    MoveL Offs(pOrigin,70.60,28.59,0.00),v40,z0,tPen\WObj:=wPaper;
    MoveL Offs(pOrigin,71.45,28.80,0.00),v40,fine,tPen\WObj:=wPaper;
    MoveL Offs(pOrigin,71.45,28.80,6.00),v60,z5,tPen\WObj:=wPaper;
    MoveL Offs(pOrigin,63.80,32.84,6.00),vTravel,z5,tPen\WObj:=wPaper;
    MoveL Offs(pOrigin,63.80,32.84,0.00),v60,z0,tPen\WObj:=wPaper;
    MoveL Offs(pOrigin,62.21,28.38,0.00),v40,z0,tPen\WObj:=wPaper;
    MoveL Offs(pOrigin,62.21,26.25,0.00),v40,z0,tPen\WObj:=wPaper;
    MoveL Offs(pOrigin,62.81,24.44,0.00),v40,z0,tPen\WObj:=wPaper;
    MoveL Offs(pOrigin,63.73,23.27,0.00),v40,z0,tPen\WObj:=wPaper;
    MoveL Offs(pOrigin,63.87,22.74,0.00),v40,z0,tPen\WObj:=wPaper;
    MoveL Offs(pOrigin,63.59,22.46,0.00),v40,z0,tPen\WObj:=wPaper;
    MoveL Offs(pOrigin,61.99,22.39,0.00),v40,z0,tPen\WObj:=wPaper;
    MoveL Offs(pOrigin,61.36,23.38,0.00),v40,z0,tPen\WObj:=wPaper;
    MoveL Offs(pOrigin,60.54,23.91,0.00),v40,z0,tPen\WObj:=wPaper;
    MoveL Offs(pOrigin,60.08,25.93,0.00),v40,z0,tPen\WObj:=wPaper;
    MoveL Offs(pOrigin,60.40,28.69,0.00),v40,z0,tPen\WObj:=wPaper;
    MoveL Offs(pOrigin,60.40,28.69,0.00),v40,z0,tPen\WObj:=wPaper;
    MoveL Offs(pOrigin,60.93,29.01,0.00),v40,z0,tPen\WObj:=wPaper;
    MoveL Offs(pOrigin,63.27,32.73,0.00),v40,z0,tPen\WObj:=wPaper;
    MoveL Offs(pOrigin,65.29,34.75,0.00),v40,z0,tPen\WObj:=wPaper;
    MoveL Offs(pOrigin,65.50,35.49,0.00),v40,z0,tPen\WObj:=wPaper;
    MoveL Offs(pOrigin,65.50,35.49,0.00),v40,z0,tPen\WObj:=wPaper;
    MoveL Offs(pOrigin,63.06,34.22,0.00),v40,z0,tPen\WObj:=wPaper;
    MoveL Offs(pOrigin,61.57,32.84,0.00),v40,z0,tPen\WObj:=wPaper;
    MoveL Offs(pOrigin,60.61,30.82,0.00),v40,z0,tPen\WObj:=wPaper;
    MoveL Offs(pOrigin,60.40,28.69,0.00),v40,fine,tPen\WObj:=wPaper;
    MoveL Offs(pOrigin,60.40,28.69,6.00),v60,z5,tPen\WObj:=wPaper;
    MoveL Offs(pOrigin,57.11,24.55,6.00),vTravel,z5,tPen\WObj:=wPaper;
    MoveL Offs(pOrigin,57.11,24.55,0.00),v60,z0,tPen\WObj:=wPaper;
    MoveL Offs(pOrigin,57.67,22.00,0.00),v40,z0,tPen\WObj:=wPaper;
    MoveL Offs(pOrigin,58.91,22.00,0.00),v40,fine,tPen\WObj:=wPaper;
    MoveL Offs(pOrigin,58.91,22.00,6.00),v60,z5,tPen\WObj:=wPaper;
    MoveL Offs(pOrigin,57.64,21.89,6.00),vTravel,z5,tPen\WObj:=wPaper;
    MoveL Offs(pOrigin,57.64,21.89,0.00),v60,z0,tPen\WObj:=wPaper;
    MoveL Offs(pOrigin,56.58,21.89,0.00),v40,z0,tPen\WObj:=wPaper;
    MoveL Offs(pOrigin,56.26,22.85,0.00),v40,z0,tPen\WObj:=wPaper;
    MoveL Offs(pOrigin,55.76,23.10,0.00),v40,z0,tPen\WObj:=wPaper;
    MoveL Offs(pOrigin,55.30,24.23,0.00),v40,z0,tPen\WObj:=wPaper;
    MoveL Offs(pOrigin,55.41,24.87,0.00),v40,z0,tPen\WObj:=wPaper;
    MoveL Offs(pOrigin,56.15,24.87,0.00),v40,fine,tPen\WObj:=wPaper;
    MoveL Offs(pOrigin,56.15,24.87,6.00),v60,z5,tPen\WObj:=wPaper;
    MoveL Offs(pOrigin,53.49,30.29,6.00),vTravel,z5,tPen\WObj:=wPaper;
    MoveL Offs(pOrigin,53.49,30.29,0.00),v60,z0,tPen\WObj:=wPaper;
    MoveL Offs(pOrigin,52.86,28.59,0.00),v40,z0,tPen\WObj:=wPaper;
    MoveL Offs(pOrigin,52.54,26.25,0.00),v40,z0,tPen\WObj:=wPaper;
    MoveL Offs(pOrigin,53.03,24.23,0.00),v40,z0,tPen\WObj:=wPaper;
    MoveL Offs(pOrigin,53.88,23.06,0.00),v40,z0,tPen\WObj:=wPaper;
    MoveL Offs(pOrigin,54.03,22.32,0.00),v40,z0,tPen\WObj:=wPaper;
    MoveL Offs(pOrigin,50.84,22.74,0.00),v40,z0,tPen\WObj:=wPaper;
    MoveL Offs(pOrigin,48.39,24.02,0.00),v40,z0,tPen\WObj:=wPaper;
    MoveL Offs(pOrigin,46.94,25.72,0.00),v40,z0,tPen\WObj:=wPaper;
    MoveL Offs(pOrigin,46.59,28.27,0.00),v40,z0,tPen\WObj:=wPaper;
    MoveL Offs(pOrigin,47.26,28.91,0.00),v40,z0,tPen\WObj:=wPaper;
    MoveL Offs(pOrigin,49.99,34.86,0.00),v40,z0,tPen\WObj:=wPaper;
    MoveL Offs(pOrigin,50.31,34.86,0.00),v40,z0,tPen\WObj:=wPaper;
    MoveL Offs(pOrigin,51.05,35.60,0.00),v40,z0,tPen\WObj:=wPaper;
    MoveL Offs(pOrigin,50.31,34.86,0.00),v40,fine,tPen\WObj:=wPaper;
    MoveL Offs(pOrigin,50.31,34.86,6.00),v60,z5,tPen\WObj:=wPaper;
    MoveL Offs(pOrigin,49.24,35.92,6.00),vTravel,z5,tPen\WObj:=wPaper;
    MoveL Offs(pOrigin,49.24,35.92,0.00),v60,z0,tPen\WObj:=wPaper;
    MoveL Offs(pOrigin,46.59,30.29,0.00),v40,z0,tPen\WObj:=wPaper;
    MoveL Offs(pOrigin,46.59,28.48,0.00),v40,fine,tPen\WObj:=wPaper;
    MoveL Offs(pOrigin,46.59,28.48,6.00),v60,z5,tPen\WObj:=wPaper;
    MoveL Offs(pOrigin,46.48,30.29,6.00),vTravel,z5,tPen\WObj:=wPaper;
    MoveL Offs(pOrigin,46.48,30.29,0.00),v60,z0,tPen\WObj:=wPaper;
    MoveL Offs(pOrigin,46.09,30.61,0.00),v40,z0,tPen\WObj:=wPaper;
    MoveL Offs(pOrigin,45.10,34.22,0.00),v40,z0,tPen\WObj:=wPaper;
    MoveL Offs(pOrigin,45.10,38.04,0.00),v40,z0,tPen\WObj:=wPaper;
    MoveL Offs(pOrigin,45.70,39.85,0.00),v40,z0,tPen\WObj:=wPaper;
    MoveL Offs(pOrigin,47.90,43.57,0.00),v40,z0,tPen\WObj:=wPaper;
    MoveL Offs(pOrigin,49.21,46.76,0.00),v40,z0,tPen\WObj:=wPaper;
    MoveL Offs(pOrigin,52.01,49.84,0.00),v40,fine,tPen\WObj:=wPaper;
    MoveL Offs(pOrigin,52.01,49.84,6.00),v60,z5,tPen\WObj:=wPaper;
    MoveL Offs(pOrigin,53.17,43.46,6.00),vTravel,z5,tPen\WObj:=wPaper;
    MoveL Offs(pOrigin,53.17,43.46,0.00),v60,z0,tPen\WObj:=wPaper;
    MoveL Offs(pOrigin,48.18,39.11,0.00),v40,z0,tPen\WObj:=wPaper;
    MoveL Offs(pOrigin,46.38,36.13,0.00),v40,fine,tPen\WObj:=wPaper;
    MoveL Offs(pOrigin,46.38,36.13,6.00),v60,z5,tPen\WObj:=wPaper;
    MoveL Offs(pOrigin,48.39,39.42,6.00),vTravel,z5,tPen\WObj:=wPaper;
    MoveL Offs(pOrigin,48.39,39.42,0.00),v60,z0,tPen\WObj:=wPaper;
    MoveL Offs(pOrigin,49.35,40.38,0.00),v40,z0,tPen\WObj:=wPaper;
    MoveL Offs(pOrigin,48.39,39.42,0.00),v40,fine,tPen\WObj:=wPaper;
    MoveL Offs(pOrigin,48.39,39.42,6.00),v60,z5,tPen\WObj:=wPaper;
  ENDPROC

  PROC DrawPart27()
    MoveL Offs(pOrigin,48.18,41.23,6.00),vTravel,z5,tPen\WObj:=wPaper;
    MoveL Offs(pOrigin,48.18,41.23,0.00),v60,z0,tPen\WObj:=wPaper;
    MoveL Offs(pOrigin,50.20,43.36,0.00),v40,z0,tPen\WObj:=wPaper;
    MoveL Offs(pOrigin,52.64,45.20,0.00),v40,z0,tPen\WObj:=wPaper;
    MoveL Offs(pOrigin,55.41,46.69,0.00),v40,z0,tPen\WObj:=wPaper;
    MoveL Offs(pOrigin,58.28,47.71,0.00),v40,fine,tPen\WObj:=wPaper;
    MoveL Offs(pOrigin,58.28,47.71,6.00),v60,z5,tPen\WObj:=wPaper;
    MoveL Offs(pOrigin,54.45,42.72,6.00),vTravel,z5,tPen\WObj:=wPaper;
    MoveL Offs(pOrigin,54.45,42.72,0.00),v60,z0,tPen\WObj:=wPaper;
    MoveL Offs(pOrigin,54.98,43.25,0.00),v40,z0,tPen\WObj:=wPaper;
    MoveL Offs(pOrigin,54.45,42.72,0.00),v40,fine,tPen\WObj:=wPaper;
    MoveL Offs(pOrigin,54.45,42.72,6.00),v60,z5,tPen\WObj:=wPaper;
    MoveL Offs(pOrigin,57.32,39.96,6.00),vTravel,z5,tPen\WObj:=wPaper;
    MoveL Offs(pOrigin,57.32,39.96,0.00),v60,z0,tPen\WObj:=wPaper;
    MoveL Offs(pOrigin,60.08,42.01,0.00),v40,z0,tPen\WObj:=wPaper;
    MoveL Offs(pOrigin,63.80,43.71,0.00),v40,z0,tPen\WObj:=wPaper;
    MoveL Offs(pOrigin,64.12,44.21,0.00),v40,fine,tPen\WObj:=wPaper;
    MoveL Offs(pOrigin,64.12,44.21,6.00),v60,z5,tPen\WObj:=wPaper;
    MoveL Offs(pOrigin,72.30,46.97,6.00),vTravel,z5,tPen\WObj:=wPaper;
    MoveL Offs(pOrigin,72.30,46.97,0.00),v60,z0,tPen\WObj:=wPaper;
    MoveL Offs(pOrigin,76.34,42.93,0.00),v40,fine,tPen\WObj:=wPaper;
    MoveL Offs(pOrigin,76.34,42.93,6.00),v60,z5,tPen\WObj:=wPaper;
    MoveL Offs(pOrigin,76.76,45.06,6.00),vTravel,z5,tPen\WObj:=wPaper;
    MoveL Offs(pOrigin,76.76,45.06,0.00),v60,z0,tPen\WObj:=wPaper;
    MoveL Offs(pOrigin,76.34,45.48,0.00),v40,z0,tPen\WObj:=wPaper;
    MoveL Offs(pOrigin,76.76,45.06,0.00),v40,z0,tPen\WObj:=wPaper;
    MoveL Offs(pOrigin,76.02,45.91,0.00),v40,z0,tPen\WObj:=wPaper;
    MoveL Offs(pOrigin,75.28,46.65,0.00),v40,z0,tPen\WObj:=wPaper;
    MoveL Offs(pOrigin,76.02,45.91,0.00),v40,fine,tPen\WObj:=wPaper;
    MoveL Offs(pOrigin,76.02,45.91,6.00),v60,z5,tPen\WObj:=wPaper;
    MoveL Offs(pOrigin,76.76,36.98,6.00),vTravel,z5,tPen\WObj:=wPaper;
    MoveL Offs(pOrigin,76.76,36.98,0.00),v60,z0,tPen\WObj:=wPaper;
    MoveL Offs(pOrigin,78.46,37.30,0.00),v40,z0,tPen\WObj:=wPaper;
    MoveL Offs(pOrigin,78.89,36.98,0.00),v40,fine,tPen\WObj:=wPaper;
    MoveL Offs(pOrigin,78.89,36.98,6.00),v60,z5,tPen\WObj:=wPaper;
    MoveL Offs(pOrigin,81.54,37.09,6.00),vTravel,z5,tPen\WObj:=wPaper;
    MoveL Offs(pOrigin,81.54,37.09,0.00),v60,z0,tPen\WObj:=wPaper;
    MoveL Offs(pOrigin,83.56,36.98,0.00),v40,z0,tPen\WObj:=wPaper;
    MoveL Offs(pOrigin,83.56,36.98,0.00),v40,z0,tPen\WObj:=wPaper;
    MoveL Offs(pOrigin,83.24,36.24,0.00),v40,z0,tPen\WObj:=wPaper;
    MoveL Offs(pOrigin,81.76,35.17,0.00),v40,z0,tPen\WObj:=wPaper;
    MoveL Offs(pOrigin,81.65,34.54,0.00),v40,z0,tPen\WObj:=wPaper;
    MoveL Offs(pOrigin,80.59,32.84,0.00),v40,fine,tPen\WObj:=wPaper;
    MoveL Offs(pOrigin,80.59,32.84,6.00),v60,z5,tPen\WObj:=wPaper;
    MoveL Offs(pOrigin,83.56,36.98,6.00),vTravel,z5,tPen\WObj:=wPaper;
    MoveL Offs(pOrigin,83.56,36.98,0.00),v60,z0,tPen\WObj:=wPaper;
    MoveL Offs(pOrigin,84.94,37.72,0.00),v40,z0,tPen\WObj:=wPaper;
    MoveL Offs(pOrigin,85.37,38.58,0.00),v40,z0,tPen\WObj:=wPaper;
    MoveL Offs(pOrigin,85.37,38.58,0.00),v40,z0,tPen\WObj:=wPaper;
    MoveL Offs(pOrigin,84.52,39.21,0.00),v40,z0,tPen\WObj:=wPaper;
    MoveL Offs(pOrigin,85.37,38.58,0.00),v40,z0,tPen\WObj:=wPaper;
    MoveL Offs(pOrigin,86.01,38.79,0.00),v40,z0,tPen\WObj:=wPaper;
    MoveL Offs(pOrigin,88.34,40.84,0.00),v40,z0,tPen\WObj:=wPaper;
    MoveL Offs(pOrigin,90.68,41.44,0.00),v40,fine,tPen\WObj:=wPaper;
    MoveL Offs(pOrigin,90.68,41.44,6.00),v60,z5,tPen\WObj:=wPaper;
    MoveL Offs(pOrigin,93.12,40.91,6.00),vTravel,z5,tPen\WObj:=wPaper;
    MoveL Offs(pOrigin,93.12,40.91,0.00),v60,z0,tPen\WObj:=wPaper;
    MoveL Offs(pOrigin,93.76,40.74,0.00),v40,z0,tPen\WObj:=wPaper;
    MoveL Offs(pOrigin,94.61,41.66,0.00),v40,fine,tPen\WObj:=wPaper;
    MoveL Offs(pOrigin,94.61,41.66,6.00),v60,z5,tPen\WObj:=wPaper;
    MoveL Offs(pOrigin,93.87,40.70,6.00),vTravel,z5,tPen\WObj:=wPaper;
    MoveL Offs(pOrigin,93.87,40.70,0.00),v60,z0,tPen\WObj:=wPaper;
    MoveL Offs(pOrigin,96.10,39.85,0.00),v40,z0,tPen\WObj:=wPaper;
    MoveL Offs(pOrigin,96.95,40.59,0.00),v40,z0,tPen\WObj:=wPaper;
    MoveL Offs(pOrigin,96.53,41.02,0.00),v40,z0,tPen\WObj:=wPaper;
    MoveL Offs(pOrigin,96.95,40.59,0.00),v40,z0,tPen\WObj:=wPaper;
    MoveL Offs(pOrigin,96.10,41.34,0.00),v40,z0,tPen\WObj:=wPaper;
    MoveL Offs(pOrigin,95.78,41.66,0.00),v40,z0,tPen\WObj:=wPaper;
    MoveL Offs(pOrigin,96.10,41.34,0.00),v40,fine,tPen\WObj:=wPaper;
    MoveL Offs(pOrigin,96.10,41.34,6.00),v60,z5,tPen\WObj:=wPaper;
    MoveL Offs(pOrigin,88.13,44.10,6.00),vTravel,z5,tPen\WObj:=wPaper;
    MoveL Offs(pOrigin,88.13,44.10,0.00),v60,z0,tPen\WObj:=wPaper;
    MoveL Offs(pOrigin,87.81,44.42,0.00),v40,z0,tPen\WObj:=wPaper;
    MoveL Offs(pOrigin,88.13,44.10,0.00),v40,z0,tPen\WObj:=wPaper;
    MoveL Offs(pOrigin,87.49,44.63,0.00),v40,z0,tPen\WObj:=wPaper;
    MoveL Offs(pOrigin,86.96,45.16,0.00),v40,z0,tPen\WObj:=wPaper;
    MoveL Offs(pOrigin,87.49,44.63,0.00),v40,fine,tPen\WObj:=wPaper;
    MoveL Offs(pOrigin,87.49,44.63,6.00),v60,z5,tPen\WObj:=wPaper;
    MoveL Offs(pOrigin,86.22,38.89,6.00),vTravel,z5,tPen\WObj:=wPaper;
    MoveL Offs(pOrigin,86.22,38.89,0.00),v60,z0,tPen\WObj:=wPaper;
    MoveL Offs(pOrigin,87.07,39.74,0.00),v40,z0,tPen\WObj:=wPaper;
    MoveL Offs(pOrigin,86.22,38.89,0.00),v40,fine,tPen\WObj:=wPaper;
    MoveL Offs(pOrigin,86.22,38.89,6.00),v60,z5,tPen\WObj:=wPaper;
    MoveL Offs(pOrigin,84.09,37.51,6.00),vTravel,z5,tPen\WObj:=wPaper;
    MoveL Offs(pOrigin,84.09,37.51,0.00),v60,z0,tPen\WObj:=wPaper;
    MoveL Offs(pOrigin,83.35,38.29,0.00),v40,z0,tPen\WObj:=wPaper;
    MoveL Offs(pOrigin,81.33,39.21,0.00),v40,z0,tPen\WObj:=wPaper;
    MoveL Offs(pOrigin,78.99,39.74,0.00),v40,z0,tPen\WObj:=wPaper;
    MoveL Offs(pOrigin,76.23,39.74,0.00),v40,z0,tPen\WObj:=wPaper;
    MoveL Offs(pOrigin,71.24,38.40,0.00),v40,z0,tPen\WObj:=wPaper;
    MoveL Offs(pOrigin,65.50,35.49,0.00),v40,fine,tPen\WObj:=wPaper;
    MoveL Offs(pOrigin,65.50,35.49,6.00),v60,z5,tPen\WObj:=wPaper;
    MoveL Offs(pOrigin,48.08,24.23,6.00),vTravel,z5,tPen\WObj:=wPaper;
    MoveL Offs(pOrigin,48.08,24.23,0.00),v60,z0,tPen\WObj:=wPaper;
    MoveL Offs(pOrigin,47.65,24.66,0.00),v40,z0,tPen\WObj:=wPaper;
    MoveL Offs(pOrigin,48.08,24.23,0.00),v40,fine,tPen\WObj:=wPaper;
    MoveL Offs(pOrigin,48.08,24.23,6.00),v60,z5,tPen\WObj:=wPaper;
    MoveL Offs(pOrigin,98.33,12.86,6.00),vTravel,z5,tPen\WObj:=wPaper;
    MoveL Offs(pOrigin,98.33,12.86,0.00),v60,z0,tPen\WObj:=wPaper;
    MoveL Offs(pOrigin,97.91,12.01,0.00),v40,z0,tPen\WObj:=wPaper;
    MoveL Offs(pOrigin,97.91,11.06,0.00),v40,fine,tPen\WObj:=wPaper;
    MoveL Offs(pOrigin,97.91,11.06,6.00),v60,z5,tPen\WObj:=wPaper;
    MoveL Offs(pOrigin,90.47,54.83,6.00),vTravel,z5,tPen\WObj:=wPaper;
    MoveL Offs(pOrigin,90.47,54.83,0.00),v60,z0,tPen\WObj:=wPaper;
    MoveL Offs(pOrigin,92.91,57.28,0.00),v40,z0,tPen\WObj:=wPaper;
    MoveL Offs(pOrigin,90.47,54.83,0.00),v40,fine,tPen\WObj:=wPaper;
    MoveL Offs(pOrigin,90.47,54.83,6.00),v60,z5,tPen\WObj:=wPaper;
    MoveL Offs(pOrigin,97.48,140.36,6.00),vTravel,z5,tPen\WObj:=wPaper;
    MoveL Offs(pOrigin,97.48,140.36,0.00),v60,z0,tPen\WObj:=wPaper;
    MoveL Offs(pOrigin,97.16,141.00,0.00),v40,z0,tPen\WObj:=wPaper;
    MoveL Offs(pOrigin,97.38,141.43,0.00),v40,z0,tPen\WObj:=wPaper;
    MoveL Offs(pOrigin,97.38,141.43,0.00),v40,z0,tPen\WObj:=wPaper;
    MoveL Offs(pOrigin,98.44,142.17,0.00),v40,z0,tPen\WObj:=wPaper;
    MoveL Offs(pOrigin,98.65,143.02,0.00),v40,z0,tPen\WObj:=wPaper;
    MoveL Offs(pOrigin,98.65,143.02,0.00),v40,z0,tPen\WObj:=wPaper;
    MoveL Offs(pOrigin,98.33,143.34,0.00),v40,z0,tPen\WObj:=wPaper;
    MoveL Offs(pOrigin,99.29,145.25,0.00),v40,fine,tPen\WObj:=wPaper;
    MoveL Offs(pOrigin,99.29,145.25,6.00),v60,z5,tPen\WObj:=wPaper;
    MoveL Offs(pOrigin,97.80,144.51,6.00),vTravel,z5,tPen\WObj:=wPaper;
    MoveL Offs(pOrigin,97.80,144.51,0.00),v60,z0,tPen\WObj:=wPaper;
  ENDPROC

  PROC DrawPart28()
    MoveL Offs(pOrigin,99.61,148.23,0.00),v40,z0,tPen\WObj:=wPaper;
    MoveL Offs(pOrigin,99.82,148.33,0.00),v40,z0,tPen\WObj:=wPaper;
    MoveL Offs(pOrigin,99.61,148.54,0.00),v40,z0,tPen\WObj:=wPaper;
    MoveL Offs(pOrigin,100.24,148.97,0.00),v40,z0,tPen\WObj:=wPaper;
    MoveL Offs(pOrigin,100.24,148.97,0.00),v40,z0,tPen\WObj:=wPaper;
    MoveL Offs(pOrigin,101.73,150.88,0.00),v40,fine,tPen\WObj:=wPaper;
    MoveL Offs(pOrigin,101.73,150.88,6.00),v60,z5,tPen\WObj:=wPaper;
    MoveL Offs(pOrigin,100.35,150.77,6.00),vTravel,z5,tPen\WObj:=wPaper;
    MoveL Offs(pOrigin,100.35,150.77,0.00),v60,z0,tPen\WObj:=wPaper;
    MoveL Offs(pOrigin,98.97,149.39,0.00),v40,z0,tPen\WObj:=wPaper;
    MoveL Offs(pOrigin,97.16,146.42,0.00),v40,z0,tPen\WObj:=wPaper;
    MoveL Offs(pOrigin,97.16,146.42,0.00),v40,z0,tPen\WObj:=wPaper;
    MoveL Offs(pOrigin,97.38,146.21,0.00),v40,z0,tPen\WObj:=wPaper;
    MoveL Offs(pOrigin,97.16,144.29,0.00),v40,fine,tPen\WObj:=wPaper;
    MoveL Offs(pOrigin,97.16,144.29,6.00),v60,z5,tPen\WObj:=wPaper;
    MoveL Offs(pOrigin,96.63,142.59,6.00),vTravel,z5,tPen\WObj:=wPaper;
    MoveL Offs(pOrigin,96.63,142.59,0.00),v60,z0,tPen\WObj:=wPaper;
    MoveL Offs(pOrigin,96.70,141.74,0.00),v40,z0,tPen\WObj:=wPaper;
    MoveL Offs(pOrigin,97.16,141.43,0.00),v40,z0,tPen\WObj:=wPaper;
    MoveL Offs(pOrigin,97.38,141.43,0.00),v40,z0,tPen\WObj:=wPaper;
    MoveL Offs(pOrigin,98.76,141.00,0.00),v40,z0,tPen\WObj:=wPaper;
    MoveL Offs(pOrigin,98.76,140.68,0.00),v40,z0,tPen\WObj:=wPaper;
    MoveL Offs(pOrigin,99.00,140.79,0.00),v40,z0,tPen\WObj:=wPaper;
    MoveL Offs(pOrigin,99.18,140.04,0.00),v40,z0,tPen\WObj:=wPaper;
    MoveL Offs(pOrigin,98.54,139.30,0.00),v40,z0,tPen\WObj:=wPaper;
    MoveL Offs(pOrigin,98.33,140.36,0.00),v40,fine,tPen\WObj:=wPaper;
    MoveL Offs(pOrigin,98.33,140.36,6.00),v60,z5,tPen\WObj:=wPaper;
    MoveL Offs(pOrigin,97.69,142.59,6.00),vTravel,z5,tPen\WObj:=wPaper;
    MoveL Offs(pOrigin,97.69,142.59,0.00),v60,z0,tPen\WObj:=wPaper;
    MoveL Offs(pOrigin,96.63,142.59,0.00),v40,fine,tPen\WObj:=wPaper;
    MoveL Offs(pOrigin,96.63,142.59,6.00),v60,z5,tPen\WObj:=wPaper;
    MoveL Offs(pOrigin,98.65,143.02,6.00),vTravel,z5,tPen\WObj:=wPaper;
    MoveL Offs(pOrigin,98.65,143.02,0.00),v60,z0,tPen\WObj:=wPaper;
    MoveL Offs(pOrigin,100.99,145.68,0.00),v40,z0,tPen\WObj:=wPaper;
    MoveL Offs(pOrigin,100.99,145.68,0.00),v40,z0,tPen\WObj:=wPaper;
    MoveL Offs(pOrigin,101.84,147.38,0.00),v40,z0,tPen\WObj:=wPaper;
    MoveL Offs(pOrigin,101.84,147.38,0.00),v40,z0,tPen\WObj:=wPaper;
    MoveL Offs(pOrigin,101.52,148.65,0.00),v40,fine,tPen\WObj:=wPaper;
    MoveL Offs(pOrigin,101.52,148.65,6.00),v60,z5,tPen\WObj:=wPaper;
    MoveL Offs(pOrigin,97.16,146.42,6.00),vTravel,z5,tPen\WObj:=wPaper;
    MoveL Offs(pOrigin,97.16,146.42,0.00),v60,z0,tPen\WObj:=wPaper;
    MoveL Offs(pOrigin,95.89,145.68,0.00),v40,fine,tPen\WObj:=wPaper;
    MoveL Offs(pOrigin,95.89,145.68,6.00),v60,z5,tPen\WObj:=wPaper;
    MoveL Offs(pOrigin,96.63,150.03,6.00),vTravel,z5,tPen\WObj:=wPaper;
    MoveL Offs(pOrigin,96.63,150.03,0.00),v60,z0,tPen\WObj:=wPaper;
    MoveL Offs(pOrigin,96.21,150.88,0.00),v40,z0,tPen\WObj:=wPaper;
    MoveL Offs(pOrigin,96.21,152.26,0.00),v40,z0,tPen\WObj:=wPaper;
    MoveL Offs(pOrigin,96.21,152.26,0.00),v40,z0,tPen\WObj:=wPaper;
    MoveL Offs(pOrigin,96.77,152.58,0.00),v40,z0,tPen\WObj:=wPaper;
    MoveL Offs(pOrigin,97.59,154.60,0.00),v40,z0,tPen\WObj:=wPaper;
    MoveL Offs(pOrigin,97.59,154.60,0.00),v40,z0,tPen\WObj:=wPaper;
    MoveL Offs(pOrigin,99.50,156.02,0.00),v40,z0,tPen\WObj:=wPaper;
    MoveL Offs(pOrigin,103.40,156.94,0.00),v40,z0,tPen\WObj:=wPaper;
    MoveL Offs(pOrigin,103.01,157.40,0.00),v40,z0,tPen\WObj:=wPaper;
    MoveL Offs(pOrigin,101.84,157.68,0.00),v40,fine,tPen\WObj:=wPaper;
    MoveL Offs(pOrigin,101.84,157.68,6.00),v60,z5,tPen\WObj:=wPaper;
    MoveL Offs(pOrigin,105.13,156.51,6.00),vTravel,z5,tPen\WObj:=wPaper;
    MoveL Offs(pOrigin,105.13,156.51,0.00),v60,z0,tPen\WObj:=wPaper;
    MoveL Offs(pOrigin,109.17,156.30,0.00),v40,fine,tPen\WObj:=wPaper;
    MoveL Offs(pOrigin,109.17,156.30,6.00),v60,z5,tPen\WObj:=wPaper;
    MoveL Offs(pOrigin,107.89,155.66,6.00),vTravel,z5,tPen\WObj:=wPaper;
    MoveL Offs(pOrigin,107.89,155.66,0.00),v60,z0,tPen\WObj:=wPaper;
    MoveL Offs(pOrigin,105.34,155.56,0.00),v40,z0,tPen\WObj:=wPaper;
    MoveL Offs(pOrigin,104.88,155.98,0.00),v40,z0,tPen\WObj:=wPaper;
    MoveL Offs(pOrigin,105.13,156.51,0.00),v40,z0,tPen\WObj:=wPaper;
    MoveL Offs(pOrigin,105.13,156.51,0.00),v40,z0,tPen\WObj:=wPaper;
    MoveL Offs(pOrigin,103.86,157.72,0.00),v40,z0,tPen\WObj:=wPaper;
    MoveL Offs(pOrigin,101.73,158.53,0.00),v40,z0,tPen\WObj:=wPaper;
    MoveL Offs(pOrigin,99.50,158.25,0.00),v40,z0,tPen\WObj:=wPaper;
    MoveL Offs(pOrigin,98.22,157.57,0.00),v40,z0,tPen\WObj:=wPaper;
    MoveL Offs(pOrigin,97.91,157.04,0.00),v40,z0,tPen\WObj:=wPaper;
    MoveL Offs(pOrigin,97.91,157.04,0.00),v40,z0,tPen\WObj:=wPaper;
    MoveL Offs(pOrigin,96.74,156.30,0.00),v40,fine,tPen\WObj:=wPaper;
    MoveL Offs(pOrigin,96.74,156.30,6.00),v60,z5,tPen\WObj:=wPaper;
    MoveL Offs(pOrigin,97.59,154.60,6.00),vTravel,z5,tPen\WObj:=wPaper;
    MoveL Offs(pOrigin,97.59,154.60,0.00),v60,z0,tPen\WObj:=wPaper;
    MoveL Offs(pOrigin,96.84,154.18,0.00),v40,z0,tPen\WObj:=wPaper;
    MoveL Offs(pOrigin,97.27,153.86,0.00),v40,z0,tPen\WObj:=wPaper;
    MoveL Offs(pOrigin,96.21,153.64,0.00),v40,z0,tPen\WObj:=wPaper;
    MoveL Offs(pOrigin,96.21,152.26,0.00),v40,fine,tPen\WObj:=wPaper;
    MoveL Offs(pOrigin,96.21,152.26,6.00),v60,z5,tPen\WObj:=wPaper;
    MoveL Offs(pOrigin,98.44,153.01,6.00),vTravel,z5,tPen\WObj:=wPaper;
    MoveL Offs(pOrigin,98.44,153.01,0.00),v60,z0,tPen\WObj:=wPaper;
    MoveL Offs(pOrigin,98.86,153.43,0.00),v40,z0,tPen\WObj:=wPaper;
    MoveL Offs(pOrigin,98.44,153.01,0.00),v40,fine,tPen\WObj:=wPaper;
    MoveL Offs(pOrigin,98.44,153.01,6.00),v60,z5,tPen\WObj:=wPaper;
    MoveL Offs(pOrigin,99.29,162.25,6.00),vTravel,z5,tPen\WObj:=wPaper;
    MoveL Offs(pOrigin,99.29,162.25,0.00),v60,z0,tPen\WObj:=wPaper;
    MoveL Offs(pOrigin,99.71,162.68,0.00),v40,z0,tPen\WObj:=wPaper;
    MoveL Offs(pOrigin,99.29,162.25,0.00),v40,fine,tPen\WObj:=wPaper;
    MoveL Offs(pOrigin,99.29,162.25,6.00),v60,z5,tPen\WObj:=wPaper;
    MoveL Offs(pOrigin,103.01,165.44,6.00),vTravel,z5,tPen\WObj:=wPaper;
    MoveL Offs(pOrigin,103.01,165.44,0.00),v60,z0,tPen\WObj:=wPaper;
    MoveL Offs(pOrigin,104.49,165.76,0.00),v40,z0,tPen\WObj:=wPaper;
    MoveL Offs(pOrigin,104.49,165.76,0.00),v40,z0,tPen\WObj:=wPaper;
    MoveL Offs(pOrigin,104.81,166.22,0.00),v40,z0,tPen\WObj:=wPaper;
    MoveL Offs(pOrigin,107.26,166.82,0.00),v40,z0,tPen\WObj:=wPaper;
    MoveL Offs(pOrigin,108.74,166.71,0.00),v40,z0,tPen\WObj:=wPaper;
    MoveL Offs(pOrigin,108.74,166.71,0.00),v40,z0,tPen\WObj:=wPaper;
    MoveL Offs(pOrigin,110.23,166.46,0.00),v40,z0,tPen\WObj:=wPaper;
    MoveL Offs(pOrigin,111.44,165.44,0.00),v40,z0,tPen\WObj:=wPaper;
    MoveL Offs(pOrigin,111.72,163.74,0.00),v40,z0,tPen\WObj:=wPaper;
    MoveL Offs(pOrigin,110.97,162.68,0.00),v40,z0,tPen\WObj:=wPaper;
    MoveL Offs(pOrigin,110.97,162.68,0.00),v40,z0,tPen\WObj:=wPaper;
    MoveL Offs(pOrigin,110.44,161.93,0.00),v40,z0,tPen\WObj:=wPaper;
    MoveL Offs(pOrigin,110.44,161.93,0.00),v40,z0,tPen\WObj:=wPaper;
    MoveL Offs(pOrigin,110.48,160.98,0.00),v40,z0,tPen\WObj:=wPaper;
    MoveL Offs(pOrigin,111.08,160.55,0.00),v40,fine,tPen\WObj:=wPaper;
    MoveL Offs(pOrigin,111.08,160.55,6.00),v60,z5,tPen\WObj:=wPaper;
    MoveL Offs(pOrigin,111.08,159.06,6.00),vTravel,z5,tPen\WObj:=wPaper;
    MoveL Offs(pOrigin,111.08,159.06,0.00),v60,z0,tPen\WObj:=wPaper;
    MoveL Offs(pOrigin,110.34,159.13,0.00),v40,z0,tPen\WObj:=wPaper;
    MoveL Offs(pOrigin,109.38,159.81,0.00),v40,z0,tPen\WObj:=wPaper;
    MoveL Offs(pOrigin,109.17,159.70,0.00),v40,z0,tPen\WObj:=wPaper;
    MoveL Offs(pOrigin,109.38,160.98,0.00),v40,z0,tPen\WObj:=wPaper;
    MoveL Offs(pOrigin,109.38,160.98,0.00),v40,z0,tPen\WObj:=wPaper;
    MoveL Offs(pOrigin,110.02,161.93,0.00),v40,z0,tPen\WObj:=wPaper;
    MoveL Offs(pOrigin,110.02,161.93,0.00),v40,z0,tPen\WObj:=wPaper;
    MoveL Offs(pOrigin,110.44,163.52,0.00),v40,z0,tPen\WObj:=wPaper;
    MoveL Offs(pOrigin,110.34,164.69,0.00),v40,z0,tPen\WObj:=wPaper;
  ENDPROC

  PROC DrawPart29()
    MoveL Offs(pOrigin,108.74,166.71,0.00),v40,z0,tPen\WObj:=wPaper;
    MoveL Offs(pOrigin,108.53,165.65,0.00),v40,z0,tPen\WObj:=wPaper;
    MoveL Offs(pOrigin,106.94,166.61,0.00),v40,fine,tPen\WObj:=wPaper;
    MoveL Offs(pOrigin,106.94,166.61,6.00),v60,z5,tPen\WObj:=wPaper;
    MoveL Offs(pOrigin,107.47,165.12,6.00),vTravel,z5,tPen\WObj:=wPaper;
    MoveL Offs(pOrigin,107.47,165.12,0.00),v60,z0,tPen\WObj:=wPaper;
    MoveL Offs(pOrigin,106.51,165.54,0.00),v40,z0,tPen\WObj:=wPaper;
    MoveL Offs(pOrigin,104.49,165.76,0.00),v40,fine,tPen\WObj:=wPaper;
    MoveL Offs(pOrigin,104.49,165.76,6.00),v60,z5,tPen\WObj:=wPaper;
    MoveL Offs(pOrigin,103.01,165.44,6.00),vTravel,z5,tPen\WObj:=wPaper;
    MoveL Offs(pOrigin,103.01,165.44,0.00),v60,z0,tPen\WObj:=wPaper;
    MoveL Offs(pOrigin,103.43,166.39,0.00),v40,z0,tPen\WObj:=wPaper;
    MoveL Offs(pOrigin,104.92,167.24,0.00),v40,fine,tPen\WObj:=wPaper;
    MoveL Offs(pOrigin,104.92,167.24,6.00),v60,z5,tPen\WObj:=wPaper;
    MoveL Offs(pOrigin,108.96,165.44,6.00),vTravel,z5,tPen\WObj:=wPaper;
    MoveL Offs(pOrigin,108.96,165.44,0.00),v60,z0,tPen\WObj:=wPaper;
    MoveL Offs(pOrigin,109.49,164.27,0.00),v40,z0,tPen\WObj:=wPaper;
    MoveL Offs(pOrigin,109.17,161.82,0.00),v40,z0,tPen\WObj:=wPaper;
    MoveL Offs(pOrigin,109.38,160.98,0.00),v40,fine,tPen\WObj:=wPaper;
    MoveL Offs(pOrigin,109.38,160.98,6.00),v60,z5,tPen\WObj:=wPaper;
    MoveL Offs(pOrigin,109.17,159.70,6.00),vTravel,z5,tPen\WObj:=wPaper;
    MoveL Offs(pOrigin,109.17,159.70,0.00),v60,z0,tPen\WObj:=wPaper;
    MoveL Offs(pOrigin,108.67,160.05,0.00),v40,z0,tPen\WObj:=wPaper;
    MoveL Offs(pOrigin,108.43,160.98,0.00),v40,z0,tPen\WObj:=wPaper;
    MoveL Offs(pOrigin,108.64,162.57,0.00),v40,fine,tPen\WObj:=wPaper;
    MoveL Offs(pOrigin,108.64,162.57,6.00),v60,z5,tPen\WObj:=wPaper;
    MoveL Offs(pOrigin,110.97,162.68,6.00),vTravel,z5,tPen\WObj:=wPaper;
    MoveL Offs(pOrigin,110.97,162.68,0.00),v60,z0,tPen\WObj:=wPaper;
    MoveL Offs(pOrigin,111.19,164.16,0.00),v40,fine,tPen\WObj:=wPaper;
    MoveL Offs(pOrigin,111.19,164.16,6.00),v60,z5,tPen\WObj:=wPaper;
    MoveL Offs(pOrigin,112.68,162.25,6.00),vTravel,z5,tPen\WObj:=wPaper;
    MoveL Offs(pOrigin,112.68,162.25,0.00),v60,z0,tPen\WObj:=wPaper;
    MoveL Offs(pOrigin,112.99,162.68,0.00),v40,z0,tPen\WObj:=wPaper;
    MoveL Offs(pOrigin,112.68,162.25,0.00),v40,fine,tPen\WObj:=wPaper;
    MoveL Offs(pOrigin,112.68,162.25,6.00),v60,z5,tPen\WObj:=wPaper;
    MoveL Offs(pOrigin,114.59,162.46,6.00),vTravel,z5,tPen\WObj:=wPaper;
    MoveL Offs(pOrigin,114.59,162.46,0.00),v60,z0,tPen\WObj:=wPaper;
    MoveL Offs(pOrigin,114.59,163.31,0.00),v40,z0,tPen\WObj:=wPaper;
    MoveL Offs(pOrigin,115.33,165.01,0.00),v40,z0,tPen\WObj:=wPaper;
    MoveL Offs(pOrigin,115.33,166.07,0.00),v40,z0,tPen\WObj:=wPaper;
    MoveL Offs(pOrigin,114.91,167.14,0.00),v40,z0,tPen\WObj:=wPaper;
    MoveL Offs(pOrigin,113.74,167.99,0.00),v40,z0,tPen\WObj:=wPaper;
    MoveL Offs(pOrigin,113.63,168.84,0.00),v40,z0,tPen\WObj:=wPaper;
    MoveL Offs(pOrigin,115.86,167.99,0.00),v40,z0,tPen\WObj:=wPaper;
    MoveL Offs(pOrigin,116.71,166.61,0.00),v40,z0,tPen\WObj:=wPaper;
    MoveL Offs(pOrigin,116.64,165.01,0.00),v40,z0,tPen\WObj:=wPaper;
    MoveL Offs(pOrigin,115.12,162.57,0.00),v40,z0,tPen\WObj:=wPaper;
    MoveL Offs(pOrigin,115.54,163.31,0.00),v40,z0,tPen\WObj:=wPaper;
    MoveL Offs(pOrigin,115.86,163.63,0.00),v40,z0,tPen\WObj:=wPaper;
    MoveL Offs(pOrigin,115.54,163.31,0.00),v40,z0,tPen\WObj:=wPaper;
    MoveL Offs(pOrigin,115.97,162.46,0.00),v40,z0,tPen\WObj:=wPaper;
    MoveL Offs(pOrigin,117.14,163.52,0.00),v40,z0,tPen\WObj:=wPaper;
    MoveL Offs(pOrigin,118.20,163.42,0.00),v40,z0,tPen\WObj:=wPaper;
    MoveL Offs(pOrigin,119.79,165.44,0.00),v40,z0,tPen\WObj:=wPaper;
    MoveL Offs(pOrigin,119.79,165.44,0.00),v40,z0,tPen\WObj:=wPaper;
    MoveL Offs(pOrigin,120.43,166.07,0.00),v40,z0,tPen\WObj:=wPaper;
    MoveL Offs(pOrigin,120.43,167.77,0.00),v40,z0,tPen\WObj:=wPaper;
    MoveL Offs(pOrigin,119.86,169.05,0.00),v40,z0,tPen\WObj:=wPaper;
    MoveL Offs(pOrigin,118.62,169.69,0.00),v40,z0,tPen\WObj:=wPaper;
    MoveL Offs(pOrigin,118.62,169.69,0.00),v40,z0,tPen\WObj:=wPaper;
    MoveL Offs(pOrigin,116.82,170.32,0.00),v40,z0,tPen\WObj:=wPaper;
    MoveL Offs(pOrigin,111.61,170.22,0.00),v40,z0,tPen\WObj:=wPaper;
    MoveL Offs(pOrigin,110.12,169.79,0.00),v40,z0,tPen\WObj:=wPaper;
    MoveL Offs(pOrigin,108.74,170.01,0.00),v40,fine,tPen\WObj:=wPaper;
    MoveL Offs(pOrigin,108.74,170.01,6.00),v60,z5,tPen\WObj:=wPaper;
    MoveL Offs(pOrigin,112.46,171.39,6.00),vTravel,z5,tPen\WObj:=wPaper;
    MoveL Offs(pOrigin,112.46,171.39,0.00),v60,z0,tPen\WObj:=wPaper;
    MoveL Offs(pOrigin,113.84,171.18,0.00),v40,fine,tPen\WObj:=wPaper;
    MoveL Offs(pOrigin,113.84,171.18,6.00),v60,z5,tPen\WObj:=wPaper;
    MoveL Offs(pOrigin,118.62,169.69,6.00),vTravel,z5,tPen\WObj:=wPaper;
    MoveL Offs(pOrigin,118.62,169.69,0.00),v60,z0,tPen\WObj:=wPaper;
    MoveL Offs(pOrigin,119.79,167.77,0.00),v40,z0,tPen\WObj:=wPaper;
    MoveL Offs(pOrigin,119.79,165.44,0.00),v40,fine,tPen\WObj:=wPaper;
    MoveL Offs(pOrigin,119.79,165.44,6.00),v60,z5,tPen\WObj:=wPaper;
    MoveL Offs(pOrigin,117.67,162.57,6.00),vTravel,z5,tPen\WObj:=wPaper;
    MoveL Offs(pOrigin,117.67,162.57,0.00),v60,z0,tPen\WObj:=wPaper;
    MoveL Offs(pOrigin,116.39,162.04,0.00),v40,z0,tPen\WObj:=wPaper;
    MoveL Offs(pOrigin,116.07,161.93,0.00),v40,z0,tPen\WObj:=wPaper;
    MoveL Offs(pOrigin,115.44,160.55,0.00),v40,fine,tPen\WObj:=wPaper;
    MoveL Offs(pOrigin,115.44,160.55,6.00),v60,z5,tPen\WObj:=wPaper;
    MoveL Offs(pOrigin,110.97,158.53,6.00),vTravel,z5,tPen\WObj:=wPaper;
    MoveL Offs(pOrigin,110.97,158.53,0.00),v60,z0,tPen\WObj:=wPaper;
    MoveL Offs(pOrigin,111.29,158.21,0.00),v40,z0,tPen\WObj:=wPaper;
    MoveL Offs(pOrigin,110.97,158.53,0.00),v40,fine,tPen\WObj:=wPaper;
    MoveL Offs(pOrigin,110.97,158.53,6.00),v60,z5,tPen\WObj:=wPaper;
    MoveL Offs(pOrigin,111.40,157.15,6.00),vTravel,z5,tPen\WObj:=wPaper;
    MoveL Offs(pOrigin,111.40,157.15,0.00),v60,z0,tPen\WObj:=wPaper;
    MoveL Offs(pOrigin,109.38,157.89,0.00),v40,z0,tPen\WObj:=wPaper;
    MoveL Offs(pOrigin,109.38,157.89,0.00),v40,z0,tPen\WObj:=wPaper;
    MoveL Offs(pOrigin,109.42,157.26,0.00),v40,z0,tPen\WObj:=wPaper;
    MoveL Offs(pOrigin,109.81,156.87,0.00),v40,z0,tPen\WObj:=wPaper;
    MoveL Offs(pOrigin,108.11,157.26,0.00),v40,fine,tPen\WObj:=wPaper;
    MoveL Offs(pOrigin,108.11,157.26,6.00),v60,z5,tPen\WObj:=wPaper;
    MoveL Offs(pOrigin,107.26,158.11,6.00),vTravel,z5,tPen\WObj:=wPaper;
    MoveL Offs(pOrigin,107.26,158.11,0.00),v60,z0,tPen\WObj:=wPaper;
    MoveL Offs(pOrigin,107.04,159.17,0.00),v40,z0,tPen\WObj:=wPaper;
    MoveL Offs(pOrigin,108.00,158.53,0.00),v40,z0,tPen\WObj:=wPaper;
    MoveL Offs(pOrigin,107.57,158.96,0.00),v40,z0,tPen\WObj:=wPaper;
    MoveL Offs(pOrigin,108.00,158.53,0.00),v40,fine,tPen\WObj:=wPaper;
    MoveL Offs(pOrigin,108.00,158.53,6.00),v60,z5,tPen\WObj:=wPaper;
    MoveL Offs(pOrigin,124.89,162.25,6.00),vTravel,z5,tPen\WObj:=wPaper;
    MoveL Offs(pOrigin,124.89,162.25,0.00),v60,z0,tPen\WObj:=wPaper;
    MoveL Offs(pOrigin,127.02,163.63,0.00),v40,fine,tPen\WObj:=wPaper;
    MoveL Offs(pOrigin,127.02,163.63,6.00),v60,z5,tPen\WObj:=wPaper;
    MoveL Offs(pOrigin,127.02,170.64,6.00),vTravel,z5,tPen\WObj:=wPaper;
    MoveL Offs(pOrigin,127.02,170.64,0.00),v60,z0,tPen\WObj:=wPaper;
    MoveL Offs(pOrigin,125.00,171.32,0.00),v40,z0,tPen\WObj:=wPaper;
    MoveL Offs(pOrigin,124.79,171.92,0.00),v40,z0,tPen\WObj:=wPaper;
    MoveL Offs(pOrigin,124.79,171.92,0.00),v40,z0,tPen\WObj:=wPaper;
    MoveL Offs(pOrigin,126.81,171.81,0.00),v40,fine,tPen\WObj:=wPaper;
    MoveL Offs(pOrigin,126.81,171.81,6.00),v60,z5,tPen\WObj:=wPaper;
    MoveL Offs(pOrigin,132.44,156.83,6.00),vTravel,z5,tPen\WObj:=wPaper;
    MoveL Offs(pOrigin,132.44,156.83,0.00),v60,z0,tPen\WObj:=wPaper;
    MoveL Offs(pOrigin,134.14,157.15,0.00),v40,z0,tPen\WObj:=wPaper;
    MoveL Offs(pOrigin,137.01,156.51,0.00),v40,z0,tPen\WObj:=wPaper;
    MoveL Offs(pOrigin,137.01,156.09,0.00),v40,z0,tPen\WObj:=wPaper;
    MoveL Offs(pOrigin,133.71,156.30,0.00),v40,fine,tPen\WObj:=wPaper;
    MoveL Offs(pOrigin,133.71,156.30,6.00),v60,z5,tPen\WObj:=wPaper;
    MoveL Offs(pOrigin,137.01,156.09,6.00),vTravel,z5,tPen\WObj:=wPaper;
    MoveL Offs(pOrigin,137.01,156.09,0.00),v60,z0,tPen\WObj:=wPaper;
  ENDPROC

  PROC DrawPart30()
    MoveL Offs(pOrigin,137.32,155.59,0.00),v40,z0,tPen\WObj:=wPaper;
    MoveL Offs(pOrigin,138.39,155.24,0.00),v40,z0,tPen\WObj:=wPaper;
    MoveL Offs(pOrigin,138.71,154.28,0.00),v40,z0,tPen\WObj:=wPaper;
    MoveL Offs(pOrigin,139.56,153.75,0.00),v40,z0,tPen\WObj:=wPaper;
    MoveL Offs(pOrigin,138.71,154.28,0.00),v40,fine,tPen\WObj:=wPaper;
    MoveL Offs(pOrigin,138.71,154.28,6.00),v60,z5,tPen\WObj:=wPaper;
    MoveL Offs(pOrigin,145.40,153.75,6.00),vTravel,z5,tPen\WObj:=wPaper;
    MoveL Offs(pOrigin,145.40,153.75,0.00),v60,z0,tPen\WObj:=wPaper;
    MoveL Offs(pOrigin,146.57,153.43,0.00),v40,z0,tPen\WObj:=wPaper;
    MoveL Offs(pOrigin,147.21,154.03,0.00),v40,z0,tPen\WObj:=wPaper;
    MoveL Offs(pOrigin,147.84,154.07,0.00),v40,z0,tPen\WObj:=wPaper;
    MoveL Offs(pOrigin,147.10,154.07,0.00),v40,z0,tPen\WObj:=wPaper;
    MoveL Offs(pOrigin,146.53,154.81,0.00),v40,z0,tPen\WObj:=wPaper;
    MoveL Offs(pOrigin,146.78,155.66,0.00),v40,z0,tPen\WObj:=wPaper;
    MoveL Offs(pOrigin,146.46,154.92,0.00),v40,z0,tPen\WObj:=wPaper;
    MoveL Offs(pOrigin,145.72,155.17,0.00),v40,z0,tPen\WObj:=wPaper;
    MoveL Offs(pOrigin,145.51,155.77,0.00),v40,fine,tPen\WObj:=wPaper;
    MoveL Offs(pOrigin,145.51,155.77,6.00),v60,z5,tPen\WObj:=wPaper;
  ENDPROC

ENDMODULE
